(* CODESYS project XMLexample.project
   CompiledLibraryCompatibilityVersion: CODESYS V3.5 SP14 Patch 2

Project tree, tasks and I/O mapping:
  CODESYS_Control : CODESYS Control for Raspberry Pi MC SL, CODESYS GmbH, order no. 2302000009, version 4.10.0.0
    application Application
      libraries: SysFile, * (System); XML parsing and composing library, * (Open Source); Standard, 3.5.18.0 (System)
      task Task (cyclic, interval 250 ms, priority 1) calls prg_Example
      example/
        function block xml [ST]: ComposeXmlExample, FB_Init, OpenWriteClose, Parse
        program prg_Example [ST]
    SoftMotion General Axis Pool
    GPIOs_A_B : GPIOs A/B, 3S - Smart Software Solutions GmbH, version 4.10.0.0
        unmapped channels: digital inputs (GPIO0..GPIO31), digital outputs (GPIO0..GPIO31)
    Onewire
    Camera device
      <Empty>
    SPI
    I²C
*)

// CODESYS_Control/Application/example/prg_Example
PROGRAM prg_Example
VAR
    fbXml : xml;
END_VAR

fbXml();

END_PROGRAM

// CODESYS_Control/Application/example/xml
(* Демонстрирует анализ и составление XML-файлов *)
FUNCTION_BLOCK xml
VAR
    xBufferInitialised : BOOL := FALSE;
	File : FB_FileControl;
	stFileAccessMode : SysFile.ACCESS_MODE := SysFile.AM_WRITE_PLUS;
	szFilename : STRING := 'output.xml';
	
	Xml : FB_XmlControl;
	// выберите тип буфера
    Buffer : ARRAY [0..XmlPac.GVL_Param_XmlControl.MaxFileSize - 1] OF BYTE;
    // или этот тип буфера
	////Buffer : STRING(GVL_Param_XmlControl.MaxFileSize);
	
    xCreate : BOOL := TRUE;
    xParse : BOOL := FALSE; 

    Status : SysFile.SysTypes.RTS_IEC_RESULT;
    result : xmlpac.E_XmlError;
    uiParseStep : DINT := 0;
	xRead : BOOL;
    XmlFileBytesRead : __XWORD;

    i : UINT;
    sTag : STRING;
	sPara : STRING;
	sTagPara : STRING;
    
    asParsedParameter1 : ARRAY[0..7] OF STRING;
    asParsedParameter2 : ARRAY[0..7] OF STRING;
    asParsedData : ARRAY[0..7] OF STRING;
    index : USINT := 0;
END_VAR

IF xCreate THEN
	ComposeXmlExample();
	xCreate := FALSE;
END_IF;

IF xParse THEN
    Parse();
END_IF

(* Создает XML-файл *)
METHOD ComposeXmlExample : BOOL
VAR_INPUT
END_VAR
Xml.writeDocumentHeader(Header := '<?xml version="1.0" encoding="UTF-8"?>');
Xml.newTag('users');
Xml.newTag('user');
Xml.NewParameter('age', '42');
Xml.NewParameter('sex', 'male');
Xml.newTagData('John Doe');
Xml.closeTag();
Xml.newTag('user');
Xml.NewParameter('age', '39');
Xml.NewParameter('sex', 'female');
Xml.newTagData('Jane Doe');
Xml.closeTag();
Xml.closeTag();

OpenWriteClose();
END_METHOD

METHOD FB_Init : BOOL
VAR_INPUT
  bInitRetains : BOOL; // TRUE: переменные сохранения инициализируются (сброс теплый/холодный сброс)
  bInCopyCode : BOOL;  // TRUE: экземпляр будет позже скопирован в код копирования (изменение онлайн)
END_VAR
Xml.SetBuffer(	pString := ADR(Buffer),
				iSizeOf := SIZEOF(Buffer));

xBufferInitialised := TRUE;
END_METHOD

METHOD OpenWriteClose : BOOL
VAR_INPUT
END_VAR
// записать буфер в файл
File.Open(	Filename := szFilename,
			FileAccessMode := stFileAccessMode);

File.Write(	pString := ADR(Buffer),
			xml.Length );

File.Close();

Xml.ClearBuffer();
END_METHOD

ACTION Parse:
CASE uiParseStep OF
	0:  (* открыть файл с начала и прочитать в буфер *)
        (* буфер уже установлен в FB_Init *)
		result := Xml.ReadFile(sFileName := szFilename, udiNextOffset := 0, BytesRead => XmlFileBytesRead);
		IF result = E_XmlError.Ok THEN
            index := 0;
            uiParseStep := 10;
        ELSE
            uiParseStep := 99;
        END_IF
        
	
	10:	(* буфер теперь заполнен в памяти, а исходный файл закрыт. Итак, мы можем повторить это *)
		sTag := Xml.NextTag();
        IF XML.sTagsSeek = '/users/user' THEN
            XML.NextParameter(Parameter => asParsedParameter1[index]);
            XML.NextParameter(Parameter => asParsedParameter2[index]);
            asParsedData[index] := XML.GetTagData();
            index := index + 1;
        ELSIF sTag = '/users' THEN
            // done
            uiParseStep := 100;
		ELSIF XML.SearchPos >= XML.Length THEN
			uiParseStep := 100 ;
		END_IF  
	
    99: (* произошла ошибка *)
        ;
        
	100:(* Файл больше не содержит пользовательских тегов *)
        ;
END_CASE
END_ACTION

END_FUNCTION_BLOCK
